(* Schneider Machine Expert - Basic project WriteVar, file version 1.6.0.0 *)
(* ProjectInformations: Name=New project *)

HARDWARE
  Cpu 0: TM221CE16R
  EthernetConfiguration: NetworkName=M221, IpAllocationMode=FixedAddress, IpAddress=0.0.0.0, SubnetMask=0.0.0.0
  SerialLineConfiguration: Baud=Baud19200, Parity=ParityEven, DataBits=DataBits8, StopBits=StopBits1, PhysicalMedium=PhysicalMediumRs485, TransmissionMode=TransmissionModeModbusRtu, SlaveId=1, Addressing=SlaveAddressing
  MastTask: UsePeriodScanMode=false, PeriodScan=100
  FastTask: Period=255
  CpuBehavior: StartingMode=StartAsPreviousState, AutoSaveRamOnEeprom=true, WatchdogPeriod=250

SYMBOLS  (address, symbol, comment, settings)

POU New POU
  (* SectionNumber=1 *)

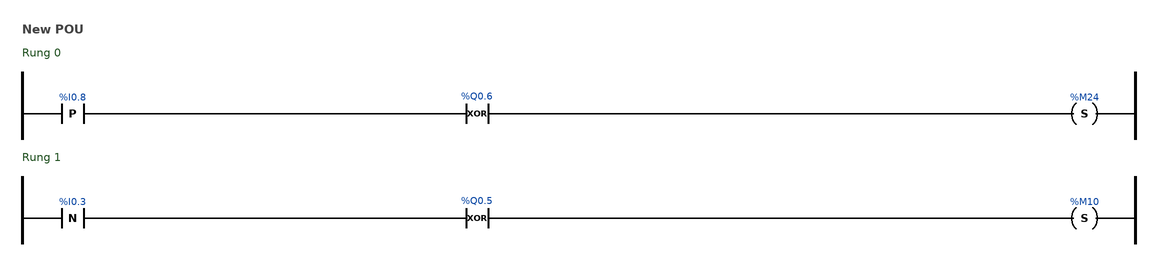

// Rung 0
  LDR %I0.8
  XOR %Q0.6
  S %M24
  // as ST:
  //   IF RISING(%I0.8) XOR %Q0.6 THEN %M24 := TRUE; END_IF;

// Rung 1
  LDF %I0.3
  XOR %Q0.5
  S %M10
  // as ST:
  //   IF FALLING(%I0.3) XOR %Q0.5 THEN %M10 := TRUE; END_IF;

// Rung 2
  BLK %WRITE_VAR0
  LDF %I0.4
  Execute
  OUT_BLK
  LD Done
  R %Q0.4
  END_BLK
  // as ST:
  //   %WRITE_VAR0(EXECUTE := FALLING(%I0.4));
  //   IF %WRITE_VAR0.Done THEN %Q0.4 := FALSE; END_IF;
  (* the ladder stored for this rung does not match its IL; not drawn *)
